FUNCTION_BLOCK Motor_Init
VAR_INPUT
	forward_start: BOOL;
	backward_start: BOOL;
END_VAR
VAR_OUTPUT
	Flag: BOOL;
END_VAR

IF forward_start OR backward_start THEN
	Flag:=TRUE;
ELSE
	Flag:=FALSE;
END_IF

END_FUNCTION_BLOCK

(* stored: Version 1.1.0.1, ProductVersion 3.1.4024.12
   POU Motor_Init: Id {a7b477bc-c74b-4d7f-9f89-ffcdb9e6f41b}, SpecialFunc None *)
